# EPICS alarm handler configuration: mps_database/bare/alarms/areas/mpln_l0b_mp03.alhConfig
GROUP NULL MPLN:L0B:MP03:1
$ALIAS MPS Link Node 53
$GUIDANCE
LTUH MPS
   Group Name: MPLN:L0B:MP03:1
   Summary PV:  MPLN:L0B:MP03:1:STATSUMY
$END
CHANNEL  MPLN:L0B:MP03:1    MPLN:L0B:MP03:1:MPS_EN_RBV		-----
CHANNEL  MPLN:L0B:MP03:1    MPLN:L0B:MP03:1:LC1_MODE_RBV		-----
